(* IEC 61131-3 sources: programs/VI-54/VI-54_20171205/VI-54_20171205/Stations/Screen/LseClass170718/Class/DiagnosticStationHandler, 1 file *)

(* ---- DiagnosticStationHandler.st ---- *)
(*!
<Class
	Name               = "DiagnosticStationHandler"
	Revision           = "1.0"
	RealtimeTask       = "false"
	CyclicTask         = "false"
	BackgroundTask     = "true"
	DefBackground      = "2 ms"
	Sigmatek           = "false"
	OSInterface        = "false"
	HighPriority       = "false"
	Automatic          = "false"
	UpdateMode         = "Prescan"
	SharedCommandTable = "true"
	Objectsize         = "(510,180)"
	Comment            = "This class login at the DiagnosticBase class. It calls every station, which is logged in at this class.">
	<Channels>
	</Channels>
	<RevDoku>
		<Owner Company="Sigmatek"/>
		<Dokumentation Revision="1.0" Date="2016-06-02" Author="HötAnt" Company="Sigmatek" Description="Creation"/>
	</RevDoku>
	<Network Name="DiagnosticStationHandler">
		<!-- List of Components in this network -->
		<Components>
			<Object
				Name       = "_base"
				Class      = "DiagnosticStationHandlerBase"
				Position   = "(240,120)"
				Visualized = "false">
				<Channels>
					<Server Name="sFuctionname"/>
					<Server Name="sStatus"/>
					<Client Name="cDiagnostic"/>
					<Client Name="cFileSys"/>
					<Client Name="cSigCLib"/>
				</Channels>
			</Object>
		</Components>
		<Comments>
		</Comments>
		<!-- List of Connections in this network -->
		<Connections>
			<Connection Source="this.sStatus" Destination="_base.sStatus" Vertices="(1358,210),(1186,210),"/>
			<Connection Source="_base.cDiagnostic" Destination="this.cDiagnostic" Vertices="(240,210),(38,210),"/>
			<Connection Source="this.sFuctionname" Destination="_base.sFuctionname" Vertices="(1358,270),(1186,270),"/>
		</Connections>
		<!-- Headerfiles -->
		<Options>
		</Options>
	</Network>
</Class>
*)
#pragma using DiagnosticStationHandlerBase

DiagnosticStationHandler : CLASS
: DiagnosticStationHandlerBase
  //Servers:
  //Clients:
  //Variables:
  //Functions:
  //Tables:
	FUNCTION @STD
		VAR_OUTPUT
			ret_code	: CONFSTATES;
		END_VAR;
	FUNCTION GLOBAL TAB @CT_;
END_CLASS;
